TYPE GearInMultiMaster_CMD_typ :
STRUCT
	StartSlave : BOOL ;
	DisengageSlave : BOOL ;
END_STRUCT
END_TYPE

(* stored: Version 1.1.0.1, ProductVersion 3.1.4024.3
   DUT GearInMultiMaster_CMD_typ: Id {6590e2f5-a2be-0012-2f9d-fcfd7f94c0fb} *)
